PROGRAM MAIN
VAR
	//st_Fupdate : ST_Event;
	btOne : BOOL := FALSE;
	
	// Trang thai cho su kien
	eEventType : E_EventType := E_EventType.Alarm;
	eEventSeverity : TcEventSeverity := TcEventSeverity.Error;
	nEventIdentity : UDINT := 32;
	sEventText : STRING(255) := 'Status';
	
	XmlPersistentEventStorage : FB_XmlPersistentEventStorage;
	EventLogger : EventLogger(XmlPersistentEventStorage);
	
END_VAR

// P_Warning();
(*
IF NOT btOne THEN
	F_UpdateEventTimestampWithSystemTime(stEvent := st_Fupdate);
	btOne := TRUE;
END_IF
*)

(*IF btOne THEN
	EventLogger.AddEvent(eEventType, eEventSeverity, nEventIdentity, sEventText);
	btOne := FALSE;
END_IF*)
Log_Csv();

END_PROGRAM

(* stored: Version 1.1.0.1, ProductVersion 3.1.4024.12
   POU MAIN: Id {34d18c9a-9e76-4259-870a-92776b81b936}, SpecialFunc None *)
